Staubli VAL3: disableQueue.pgx

public program disableQueue()
// this program disables the queing of the detected objects
begin
  // this program disables the queing of the detected objects
  //
  // Created  05-01-07                            C.CURRIVAND
  //----------------------------------------------------------------
  //
  bEnableQueuing=false
  if cfg:bLog
    logMsg(sConvNum+"(disableQueue)>>Queuing of detected object disabled")
  endIf
end
